DATA_BLOCK "EncoderET200S1COUNT_DB"   // DB87
// stored: AutoNumber true, InstanceOfName EncoderET200S1COUNT, OfSystemLibElement EncoderET200S1COUNT, OfSystemLibVersion 2.3
"EncoderET200S1COUNT"
   // VAR_INPUT
   //    EncErr : Bool;
   //    DOut_1 : Bool;
   //    DOut_2 : Bool;
   // END_VAR
   // VAR_OUTPUT
   //    DIn : Bool;
   // END_VAR
   // VAR_IN_OUT
   //    Axis : Struct
   //       Sample_T : Real;
   //       AxisType : Bool;
   //       EncoderType : Bool;
   //       Sim : Bool;
   //       AxisLimitMax : Real;
   //       AxisLimitMin : Real;
   //       MaxVelocity : Real;
   //       MaxAcceleration : Real;
   //       MaxDeceleration : Real;
   //       MonTimeTargetAppr : Real;
   //       TargetRange : Real;
   //       StandstillRange : Real;
   //       MaxFollowingDist : Real;
   //       MonitorTargetAppr : Bool;
   //       SWLimitEnable : Bool;
   //       FactorP : Real;
   //       ManVelocity : Real;
   //       ManEnable : Bool;
   //       EmergencyDec : Real;
   //       InputModuleInAddr : Int;
   //       InputModuleOutAddr : Int;
   //       InputChannelNo : Int;
   //       StepsPerRev : DInt;
   //       DisplacementPerRev : Real;
   //       NumberRevs : Int;
   //       PolarityEncoder : Int;
   //       PositionOffset : DInt;
   //       OutputModuleOutAddr : Int;
   //       OutputModuleInAddr : Int;
   //       OutputChannelNo : Int;
   //       PolarityDrive : Int;
   //       DriveInputAtMaxVel : Real;
   //       OffsetCompensation : Real;
   //       DriveInputAt100 : Real;
   //       Override : Real;
   //       ActPosition : Real;
   //       FollowingDistance : Real;
   //       RemainingDistance : Real;
   //       NomVelocity : Real;
   //       ActVelocity : Real;
   //       Sync : Bool;
   //       Error : Bool;
   //       ErrorAck : Bool;
   //       AxisState : Int;
   //       Err : Struct
   //          SWLimitMinExceeded : Bool;
   //          SWLimitMaxExceeded : Bool;
   //          TargetErr : Bool;
   //          NoSync : Bool;
   //          DirectionErr : Bool;
   //          DataErr : Bool;
   //          StartErr : Bool;
   //          DistanceErr : Bool;
   //          MasterErr : Bool;
   //          bit09 : Bool;
   //          bit10 : Bool;
   //          bit11 : Bool;
   //          bit12 : Bool;
   //          bit13 : Bool;
   //          bit14 : Bool;
   //          bit15 : Bool;
   //          StoppedMotion : Bool;
   //          EnableDriveErr : Bool;
   //          FollowingDistErr : Bool;
   //          StandstillErr : Bool;
   //          TargetApproachErr : Bool;
   //          EncoderErr : Bool;
   //          OutputErr : Bool;
   //          ConfigErr : Bool;
   //          DriveErr : Bool;
   //          bit25 : Bool;
   //          bit26 : Bool;
   //          bit27 : Bool;
   //          bit28 : Bool;
   //          bit29 : Bool;
   //          bit30 : Bool;
   //          bit31 : Bool;
   //       END_STRUCT;
   //       Config : Struct
   //          Err_AxisLimit : Bool;
   //          Err_MaxVelocity : Bool;
   //          Err_MaxAcceleration : Bool;
   //          Err_MaxDeceleration : Bool;
   //          Err_MonTimeTargetAppr : Bool;
   //          Err_TargetRange : Bool;
   //          Err_StandstillRange : Bool;
   //          Err_MaxFollowingDist : Bool;
   //          Err_EmergencyDec : Bool;
   //          Err_StepsPerRev : Bool;
   //          Err_DisplacementPerRev : Bool;
   //          Err_NumberRevs : Bool;
   //          Err_PolarityEncoder : Bool;
   //          Err_PolarityDrive : Bool;
   //          Err_DriveInputAtMaxVel : Bool;
   //          Err_AxisLength : Bool;
   //          Err_EncoderRange : Bool;
   //          Err_MaxVelRotaryAxis : Bool;
   //          Err_DriveInputAt100 : Bool;
   //       END_STRUCT;
   //       EncoderValue : DInt;
   //       RefPoint : Real;
   //       OutVelocity : Real;
   //       LastNomPosition : Real;
   //       LastNomVelocity : Real;
   //       LastNomDeceleration : Real;
   //       InternalNomPosition : Real;
   //       InternalActPos : Real;
   //       InternalPosOffset : Real;
   //       aufl : Real;
   //       AchsLaenge : Real;
   //       AchsLaenge_DI : DInt;
   //       AbsGeberLaenge_DI : DInt;
   //       LageIstwert_DI : DInt;
   //       Coord : DInt;
   //       DoneRef : Bool;
   //       EinInitLaeuft : Bool;
   //       AusInitLaeuft : Bool;
   //       EinQuittungLaeuft : Bool;
   //       AusQuittungLaeuft : Bool;
   //       EintreiberFahrbereit : Bool;
   //       ExecRef : Int;
   //       VLastNomPosition : Real;
   //       VLastNomVelocity : Real;
   //       LastInternalPosOffset : Real;
   //       RundKorrektur : Real;
   //       LastRundKorrektur : Real;
   //       LengthUnit : String[4];
   //       InputModuleType : String[24];
   //       OutputModuleType : String[24];
   //       Init : Struct
   //          I0 : Bool;
   //          I1 : Bool;
   //          I2 : Bool;
   //          I3 : Bool;
   //          I4 : Bool;
   //          I5 : Bool;
   //          I6 : Bool;
   //          I7 : Bool;
   //          I8 : Bool;
   //          I9 : Bool;
   //          I10 : Bool;
   //          I11 : Bool;
   //          I12 : Bool;
   //          I13 : Bool;
   //          I14 : Bool;
   //          I15 : Bool;
   //          I16 : Bool;
   //          I17 : Bool;
   //          I18 : Bool;
   //          I19 : Bool;
   //          I20 : Bool;
   //          I21 : Bool;
   //          I22 : Bool;
   //          I23 : Bool;
   //          I24 : Bool;
   //          I25 : Bool;
   //          I26 : Bool;
   //          I27 : Bool;
   //          I28 : Bool;
   //          I29 : Bool;
   //          I30 : Bool;
   //          I31 : Bool;
   //       END_STRUCT;
   //    END_STRUCT;
   //    Init : Bool;
   // END_VAR
   // VAR RETAIN
   //    Status : Struct
   //       STS_LOAD : Bool;
   //       ERR_LOAD : Bool;
   //       RES_STS_A : Bool;
   //       ERR_ENCODER : Bool;
   //       ERR_DO2 : Bool;
   //       ERR_PARA : Bool;
   //       ERR_DO1 : Bool;
   //       ERR_24V : Bool;
   //       STS_GATE : Bool;
   //       STS_DI : Bool;
   //       bit18 : Bool;
   //       STS_DO1 : Bool;
   //       STS_DO2 : Bool;
   //       bit21 : Bool;
   //       STS_C_UP : Bool;
   //       STS_C_DN : Bool;
   //       STS_SYN : Bool;
   //       bit09 : Bool;
   //       bit10 : Bool;
   //       STS_CMP1 : Bool;
   //       STS_CMP2 : Bool;
   //       STS_OFLW : Bool;
   //       STS_UFLW : Bool;
   //       STS_ND : Bool;
   //       byte3 : Byte;
   //    END_STRUCT;
   //    GeberAlt_DI : DInt;
   //    Addr_ActPos_DI : Int;
   //    Addr_Status : Int;
   //    Addr_LoadVal_DI : Int;
   //    Addr_Steuer : Int;
   //    Richtungsanpassung : Int;
   //    v_Faktor : Real;
   //    MaxZahl : DInt;
   //    MaxZahlHalb : DInt;
   //    PASteuer : Word;
   //    RefPointInt : Real;
   //    LoadVal_DW : DWord;
   //    EncoderZustand : Int;
   //    RefZustand : Int;
   //    aufl : Real;
   //    EncErr_alt : Bool;
   //    Taktsynchron : Bool;
   // END_VAR
BEGIN
END_DATA_BLOCK

DATA_BLOCK "IEC_Timer_0_DB"   // DB31
// stored: AutoNumber true, InstanceOfName TON_SFB, OfSystemLibElement TON, OfSystemLibVersion 1.0
"TON_SFB"
   // VAR_INPUT
   //    IN : Bool;
   //    PT : Time;
   // END_VAR
   // VAR_OUTPUT
   //    Q : Bool;
   //    ET : Time;
   // END_VAR
   // VAR RETAIN
   //    STATE : Byte;
   //    STIME : Time;
   //    ATIME : Time;
   // END_VAR
BEGIN
END_DATA_BLOCK

DATA_BLOCK "IEC_Timer_0_DB_1"   // DB60
// stored: AutoNumber true, InstanceOfName TOF_SFB, OfSystemLibElement TOF, OfSystemLibVersion 1.0
"TOF_SFB"
   // VAR_INPUT
   //    IN : Bool;
   //    PT : Time;
   // END_VAR
   // VAR_OUTPUT
   //    Q : Bool;
   //    ET : Time;
   // END_VAR
   // VAR RETAIN
   //    STATE : Byte;
   //    STIME : Time;
   //    ATIME : Time;
   // END_VAR
BEGIN
END_DATA_BLOCK

DATA_BLOCK "IEC_Timer_0_DB_3"   // DB91
// stored: AutoNumber true, InstanceOfName TON_SFB, OfSystemLibElement TON, OfSystemLibVersion 1.0
"TON_SFB"
   // VAR_INPUT
   //    IN : Bool;
   //    PT : Time;
   // END_VAR
   // VAR_OUTPUT
   //    Q : Bool;
   //    ET : Time;
   // END_VAR
   // VAR RETAIN
   //    STATE : Byte;
   //    STIME : Time;
   //    ATIME : Time;
   // END_VAR
BEGIN
END_DATA_BLOCK

DATA_BLOCK "MC_Simulation_DB"   // DB99
// stored: AutoNumber true, InstanceOfName MC_Simulation, OfSystemLibElement MC_Simulation, OfSystemLibVersion 2.1
"MC_Simulation"
   // VAR_IN_OUT
   //    Axis : Struct
   //       Sample_T : Real;
   //       AxisType : Bool;
   //       EncoderType : Bool;
   //       Sim : Bool;
   //       AxisLimitMax : Real;
   //       AxisLimitMin : Real;
   //       MaxVelocity : Real;
   //       MaxAcceleration : Real;
   //       MaxDeceleration : Real;
   //       MonTimeTargetAppr : Real;
   //       TargetRange : Real;
   //       StandstillRange : Real;
   //       MaxFollowingDist : Real;
   //       MonitorTargetAppr : Bool;
   //       SWLimitEnable : Bool;
   //       FactorP : Real;
   //       ManVelocity : Real;
   //       ManEnable : Bool;
   //       EmergencyDec : Real;
   //       InputModuleInAddr : Int;
   //       InputModuleOutAddr : Int;
   //       InputChannelNo : Int;
   //       StepsPerRev : DInt;
   //       DisplacementPerRev : Real;
   //       NumberRevs : Int;
   //       PolarityEncoder : Int;
   //       PositionOffset : DInt;
   //       OutputModuleOutAddr : Int;
   //       OutputModuleInAddr : Int;
   //       OutputChannelNo : Int;
   //       PolarityDrive : Int;
   //       DriveInputAtMaxVel : Real;
   //       OffsetCompensation : Real;
   //       DriveInputAt100 : Real;
   //       Override : Real;
   //       ActPosition : Real;
   //       FollowingDistance : Real;
   //       RemainingDistance : Real;
   //       NomVelocity : Real;
   //       ActVelocity : Real;
   //       Sync : Bool;
   //       Error : Bool;
   //       ErrorAck : Bool;
   //       AxisState : Int;
   //       Err : Struct
   //          SWLimitMinExceeded : Bool;
   //          SWLimitMaxExceeded : Bool;
   //          TargetErr : Bool;
   //          NoSync : Bool;
   //          DirectionErr : Bool;
   //          DataErr : Bool;
   //          StartErr : Bool;
   //          DistanceErr : Bool;
   //          MasterErr : Bool;
   //          bit09 : Bool;
   //          bit10 : Bool;
   //          bit11 : Bool;
   //          bit12 : Bool;
   //          bit13 : Bool;
   //          bit14 : Bool;
   //          bit15 : Bool;
   //          StoppedMotion : Bool;
   //          EnableDriveErr : Bool;
   //          FollowingDistErr : Bool;
   //          StandstillErr : Bool;
   //          TargetApproachErr : Bool;
   //          EncoderErr : Bool;
   //          OutputErr : Bool;
   //          ConfigErr : Bool;
   //          DriveErr : Bool;
   //          bit25 : Bool;
   //          bit26 : Bool;
   //          bit27 : Bool;
   //          bit28 : Bool;
   //          bit29 : Bool;
   //          bit30 : Bool;
   //          bit31 : Bool;
   //       END_STRUCT;
   //       Config : Struct
   //          Err_AxisLimit : Bool;
   //          Err_MaxVelocity : Bool;
   //          Err_MaxAcceleration : Bool;
   //          Err_MaxDeceleration : Bool;
   //          Err_MonTimeTargetAppr : Bool;
   //          Err_TargetRange : Bool;
   //          Err_StandstillRange : Bool;
   //          Err_MaxFollowingDist : Bool;
   //          Err_EmergencyDec : Bool;
   //          Err_StepsPerRev : Bool;
   //          Err_DisplacementPerRev : Bool;
   //          Err_NumberRevs : Bool;
   //          Err_PolarityEncoder : Bool;
   //          Err_PolarityDrive : Bool;
   //          Err_DriveInputAtMaxVel : Bool;
   //          Err_AxisLength : Bool;
   //          Err_EncoderRange : Bool;
   //          Err_MaxVelRotaryAxis : Bool;
   //          Err_DriveInputAt100 : Bool;
   //       END_STRUCT;
   //       EncoderValue : DInt;
   //       RefPoint : Real;
   //       OutVelocity : Real;
   //       LastNomPosition : Real;
   //       LastNomVelocity : Real;
   //       LastNomDeceleration : Real;
   //       InternalNomPosition : Real;
   //       InternalActPos : Real;
   //       InternalPosOffset : Real;
   //       aufl : Real;
   //       AchsLaenge : Real;
   //       AchsLaenge_DI : DInt;
   //       AbsGeberLaenge_DI : DInt;
   //       LageIstwert_DI : DInt;
   //       Coord : DInt;
   //       DoneRef : Bool;
   //       EinInitLaeuft : Bool;
   //       AusInitLaeuft : Bool;
   //       EinQuittungLaeuft : Bool;
   //       AusQuittungLaeuft : Bool;
   //       EintreiberFahrbereit : Bool;
   //       ExecRef : Int;
   //       VLastNomPosition : Real;
   //       VLastNomVelocity : Real;
   //       LastInternalPosOffset : Real;
   //       RundKorrektur : Real;
   //       LastRundKorrektur : Real;
   //       LengthUnit : String[4];
   //       InputModuleType : String[24];
   //       OutputModuleType : String[24];
   //       Init : Struct
   //          I0 : Bool;
   //          I1 : Bool;
   //          I2 : Bool;
   //          I3 : Bool;
   //          I4 : Bool;
   //          I5 : Bool;
   //          I6 : Bool;
   //          I7 : Bool;
   //          I8 : Bool;
   //          I9 : Bool;
   //          I10 : Bool;
   //          I11 : Bool;
   //          I12 : Bool;
   //          I13 : Bool;
   //          I14 : Bool;
   //          I15 : Bool;
   //          I16 : Bool;
   //          I17 : Bool;
   //          I18 : Bool;
   //          I19 : Bool;
   //          I20 : Bool;
   //          I21 : Bool;
   //          I22 : Bool;
   //          I23 : Bool;
   //          I24 : Bool;
   //          I25 : Bool;
   //          I26 : Bool;
   //          I27 : Bool;
   //          I28 : Bool;
   //          I29 : Bool;
   //          I30 : Bool;
   //          I31 : Bool;
   //       END_STRUCT;
   //    END_STRUCT;
   //    Init : Bool;
   // END_VAR
   // VAR RETAIN
   //    Raster : Bool;
   //    Bitanzahl : Int;
   //    LageDiff_R : Real;
   //    Faktor : Real;
   //    AusFaktor : Real;
   //    WertBei10V : Real;
   // END_VAR
BEGIN
END_DATA_BLOCK

DATA_BLOCK "Move2Done"   // DB88
// stored: AutoNumber true, InstanceOfName TON_SFB, OfSystemLibElement TON, OfSystemLibVersion 1.0
"TON_SFB"
   // VAR_INPUT
   //    IN : Bool;
   //    PT : Time;
   // END_VAR
   // VAR_OUTPUT
   //    Q : Bool;
   //    ET : Time;
   // END_VAR
   // VAR RETAIN
   //    STATE : Byte;
   //    STIME : Time;
   //    ATIME : Time;
   // END_VAR
BEGIN
END_DATA_BLOCK

DATA_BLOCK "NotEnoughProducts"   // DB84
// stored: AutoNumber true, InstanceOfName TON_SFB, OfSystemLibElement TON, OfSystemLibVersion 1.0
"TON_SFB"
   // VAR_INPUT
   //    IN : Bool;
   //    PT : Time;
   // END_VAR
   // VAR_OUTPUT
   //    Q : Bool;
   //    ET : Time;
   // END_VAR
   // VAR RETAIN
   //    STATE : Byte;
   //    STIME : Time;
   //    ATIME : Time;
   // END_VAR
BEGIN
END_DATA_BLOCK

DATA_BLOCK "OutputSinamics_DB"   // DB14
// stored: AutoNumber true, InstanceOfName OutputSinamics, OfSystemLibElement OutputSinamics, OfSystemLibVersion 2.3
"OutputSinamics"
   // VAR_INPUT
   //    TelNumber : Int;
   //    EnableDrive : Bool;
   //    StopMode : Int;
   //    OutErr : Bool;
   // END_VAR
   // VAR_OUTPUT
   //    OperationEnabled : Bool;
   //    Err_ID : Word;
   // END_VAR
   // VAR_IN_OUT
   //    Axis : Struct
   //       Sample_T : Real;
   //       AxisType : Bool;
   //       EncoderType : Bool;
   //       Sim : Bool;
   //       AxisLimitMax : Real;
   //       AxisLimitMin : Real;
   //       MaxVelocity : Real;
   //       MaxAcceleration : Real;
   //       MaxDeceleration : Real;
   //       MonTimeTargetAppr : Real;
   //       TargetRange : Real;
   //       StandstillRange : Real;
   //       MaxFollowingDist : Real;
   //       MonitorTargetAppr : Bool;
   //       SWLimitEnable : Bool;
   //       FactorP : Real;
   //       ManVelocity : Real;
   //       ManEnable : Bool;
   //       EmergencyDec : Real;
   //       InputModuleInAddr : Int;
   //       InputModuleOutAddr : Int;
   //       InputChannelNo : Int;
   //       StepsPerRev : DInt;
   //       DisplacementPerRev : Real;
   //       NumberRevs : Int;
   //       PolarityEncoder : Int;
   //       PositionOffset : DInt;
   //       OutputModuleOutAddr : Int;
   //       OutputModuleInAddr : Int;
   //       OutputChannelNo : Int;
   //       PolarityDrive : Int;
   //       DriveInputAtMaxVel : Real;
   //       OffsetCompensation : Real;
   //       DriveInputAt100 : Real;
   //       Override : Real;
   //       ActPosition : Real;
   //       FollowingDistance : Real;
   //       RemainingDistance : Real;
   //       NomVelocity : Real;
   //       ActVelocity : Real;
   //       Sync : Bool;
   //       Error : Bool;
   //       ErrorAck : Bool;
   //       AxisState : Int;
   //       Err : Struct
   //          SWLimitMinExceeded : Bool;
   //          SWLimitMaxExceeded : Bool;
   //          TargetErr : Bool;
   //          NoSync : Bool;
   //          DirectionErr : Bool;
   //          DataErr : Bool;
   //          StartErr : Bool;
   //          DistanceErr : Bool;
   //          MasterErr : Bool;
   //          bit09 : Bool;
   //          bit10 : Bool;
   //          bit11 : Bool;
   //          bit12 : Bool;
   //          bit13 : Bool;
   //          bit14 : Bool;
   //          bit15 : Bool;
   //          StoppedMotion : Bool;
   //          EnableDriveErr : Bool;
   //          FollowingDistErr : Bool;
   //          StandstillErr : Bool;
   //          TargetApproachErr : Bool;
   //          EncoderErr : Bool;
   //          OutputErr : Bool;
   //          ConfigErr : Bool;
   //          DriveErr : Bool;
   //          bit25 : Bool;
   //          bit26 : Bool;
   //          bit27 : Bool;
   //          bit28 : Bool;
   //          bit29 : Bool;
   //          bit30 : Bool;
   //          bit31 : Bool;
   //       END_STRUCT;
   //       Config : Struct
   //          Err_AxisLimit : Bool;
   //          Err_MaxVelocity : Bool;
   //          Err_MaxAcceleration : Bool;
   //          Err_MaxDeceleration : Bool;
   //          Err_MonTimeTargetAppr : Bool;
   //          Err_TargetRange : Bool;
   //          Err_StandstillRange : Bool;
   //          Err_MaxFollowingDist : Bool;
   //          Err_EmergencyDec : Bool;
   //          Err_StepsPerRev : Bool;
   //          Err_DisplacementPerRev : Bool;
   //          Err_NumberRevs : Bool;
   //          Err_PolarityEncoder : Bool;
   //          Err_PolarityDrive : Bool;
   //          Err_DriveInputAtMaxVel : Bool;
   //          Err_AxisLength : Bool;
   //          Err_EncoderRange : Bool;
   //          Err_MaxVelRotaryAxis : Bool;
   //          Err_DriveInputAt100 : Bool;
   //       END_STRUCT;
   //       EncoderValue : DInt;
   //       RefPoint : Real;
   //       OutVelocity : Real;
   //       LastNomPosition : Real;
   //       LastNomVelocity : Real;
   //       LastNomDeceleration : Real;
   //       InternalNomPosition : Real;
   //       InternalActPos : Real;
   //       InternalPosOffset : Real;
   //       aufl : Real;
   //       AchsLaenge : Real;
   //       AchsLaenge_DI : DInt;
   //       AbsGeberLaenge_DI : DInt;
   //       LageIstwert_DI : DInt;
   //       Coord : DInt;
   //       DoneRef : Bool;
   //       EinInitLaeuft : Bool;
   //       AusInitLaeuft : Bool;
   //       EinQuittungLaeuft : Bool;
   //       AusQuittungLaeuft : Bool;
   //       EintreiberFahrbereit : Bool;
   //       ExecRef : Int;
   //       VLastNomPosition : Real;
   //       VLastNomVelocity : Real;
   //       LastInternalPosOffset : Real;
   //       RundKorrektur : Real;
   //       LastRundKorrektur : Real;
   //       LengthUnit : String[4];
   //       InputModuleType : String[24];
   //       OutputModuleType : String[24];
   //       Init : Struct
   //          I0 : Bool;
   //          I1 : Bool;
   //          I2 : Bool;
   //          I3 : Bool;
   //          I4 : Bool;
   //          I5 : Bool;
   //          I6 : Bool;
   //          I7 : Bool;
   //          I8 : Bool;
   //          I9 : Bool;
   //          I10 : Bool;
   //          I11 : Bool;
   //          I12 : Bool;
   //          I13 : Bool;
   //          I14 : Bool;
   //          I15 : Bool;
   //          I16 : Bool;
   //          I17 : Bool;
   //          I18 : Bool;
   //          I19 : Bool;
   //          I20 : Bool;
   //          I21 : Bool;
   //          I22 : Bool;
   //          I23 : Bool;
   //          I24 : Bool;
   //          I25 : Bool;
   //          I26 : Bool;
   //          I27 : Bool;
   //          I28 : Bool;
   //          I29 : Bool;
   //          I30 : Bool;
   //          I31 : Bool;
   //       END_STRUCT;
   //    END_STRUCT;
   //    Init : Bool;
   // END_VAR
   // VAR RETAIN
   //    CONFIGURATION_DATA : Struct
   //       InputModuleInAddr : Int;
   //       OutputModuleOutAddr : Int;
   //       ProfiBus : Bool;
   //       ProfiNet : Bool;
   //       ID_Mastersystem : Int;
   //       Telegrammnumber : Int;
   //       TelegrFromInput : Int;
   //       InputFound : Bool;
   //       synchronous : Bool;
   //       invalid : Bool;
   //    END_STRUCT;
   //    Faktor : Real;
   //    OutputValue_R : Real;
   //    Lifecounter : Int;
   //    Addr_STW1 : Int;
   //    Addr_STW2 : Int;
   //    Addr_MRED : Int;
   //    Addr_ZSW1 : Int;
   //    Addr_ZSW2 : Int;
   //    Addr_MELDW : Int;
   //    Addr_NSOLL_B : Int;
   //    Addr_XERR : Int;
   //    Addr_KPC : Int;
   //    STW1_Offset : Int;
   //    STW2_Offset : Int;
   //    ZSW1_Offset : Int;
   //    ZSW2_Offset : Int;
   //    MRED_Offset : Int;
   //    MELDW_Offset : Int;
   //    NSOLL_B_Offset : Int;
   //    XERR_Offset : Int;
   //    KPC_Offset : Int;
   //    OutputValue : DInt;
   //    Quittungsautomat : Int;
   //    Einschaltautomat : Int;
   //    ZSW1 : Word;
   //    ZSW2 : Word;
   //    STW1 : Word;
   //    STW2 : Word;
   //    MELDW : Word;
   //    MRED : Word;
   //    wrong_OB : Bool;
   //    ERRORCODE : DWord;
   //    Virgin : Bool;
   //    FirstNormalRun : Bool;
   // END_VAR
BEGIN
END_DATA_BLOCK

DATA_BLOCK "OutputUniversal_DB"   // DB9
// stored: AutoNumber true, InstanceOfName OutputUniversal, OfSystemLibElement OutputUniversal, OfSystemLibVersion 2.1
"OutputUniversal"
   // VAR_INPUT
   //    EnableDrive : Bool;
   //    IntAtMaxVelocity : Int;
   //    OutErr : Bool;
   // END_VAR
   // VAR_OUTPUT
   //    OutputValue : Int;
   //    OutValAbs : Int;
   //    OutValSign : Bool;
   // END_VAR
   // VAR_IN_OUT
   //    Axis : Struct
   //       Sample_T : Real;
   //       AxisType : Bool;
   //       EncoderType : Bool;
   //       Sim : Bool;
   //       AxisLimitMax : Real;
   //       AxisLimitMin : Real;
   //       MaxVelocity : Real;
   //       MaxAcceleration : Real;
   //       MaxDeceleration : Real;
   //       MonTimeTargetAppr : Real;
   //       TargetRange : Real;
   //       StandstillRange : Real;
   //       MaxFollowingDist : Real;
   //       MonitorTargetAppr : Bool;
   //       SWLimitEnable : Bool;
   //       FactorP : Real;
   //       ManVelocity : Real;
   //       ManEnable : Bool;
   //       EmergencyDec : Real;
   //       InputModuleInAddr : Int;
   //       InputModuleOutAddr : Int;
   //       InputChannelNo : Int;
   //       StepsPerRev : DInt;
   //       DisplacementPerRev : Real;
   //       NumberRevs : Int;
   //       PolarityEncoder : Int;
   //       PositionOffset : DInt;
   //       OutputModuleOutAddr : Int;
   //       OutputModuleInAddr : Int;
   //       OutputChannelNo : Int;
   //       PolarityDrive : Int;
   //       DriveInputAtMaxVel : Real;
   //       OffsetCompensation : Real;
   //       DriveInputAt100 : Real;
   //       Override : Real;
   //       ActPosition : Real;
   //       FollowingDistance : Real;
   //       RemainingDistance : Real;
   //       NomVelocity : Real;
   //       ActVelocity : Real;
   //       Sync : Bool;
   //       Error : Bool;
   //       ErrorAck : Bool;
   //       AxisState : Int;
   //       Err : Struct
   //          SWLimitMinExceeded : Bool;
   //          SWLimitMaxExceeded : Bool;
   //          TargetErr : Bool;
   //          NoSync : Bool;
   //          DirectionErr : Bool;
   //          DataErr : Bool;
   //          StartErr : Bool;
   //          DistanceErr : Bool;
   //          MasterErr : Bool;
   //          bit09 : Bool;
   //          bit10 : Bool;
   //          bit11 : Bool;
   //          bit12 : Bool;
   //          bit13 : Bool;
   //          bit14 : Bool;
   //          bit15 : Bool;
   //          StoppedMotion : Bool;
   //          EnableDriveErr : Bool;
   //          FollowingDistErr : Bool;
   //          StandstillErr : Bool;
   //          TargetApproachErr : Bool;
   //          EncoderErr : Bool;
   //          OutputErr : Bool;
   //          ConfigErr : Bool;
   //          DriveErr : Bool;
   //          bit25 : Bool;
   //          bit26 : Bool;
   //          bit27 : Bool;
   //          bit28 : Bool;
   //          bit29 : Bool;
   //          bit30 : Bool;
   //          bit31 : Bool;
   //       END_STRUCT;
   //       Config : Struct
   //          Err_AxisLimit : Bool;
   //          Err_MaxVelocity : Bool;
   //          Err_MaxAcceleration : Bool;
   //          Err_MaxDeceleration : Bool;
   //          Err_MonTimeTargetAppr : Bool;
   //          Err_TargetRange : Bool;
   //          Err_StandstillRange : Bool;
   //          Err_MaxFollowingDist : Bool;
   //          Err_EmergencyDec : Bool;
   //          Err_StepsPerRev : Bool;
   //          Err_DisplacementPerRev : Bool;
   //          Err_NumberRevs : Bool;
   //          Err_PolarityEncoder : Bool;
   //          Err_PolarityDrive : Bool;
   //          Err_DriveInputAtMaxVel : Bool;
   //          Err_AxisLength : Bool;
   //          Err_EncoderRange : Bool;
   //          Err_MaxVelRotaryAxis : Bool;
   //          Err_DriveInputAt100 : Bool;
   //       END_STRUCT;
   //       EncoderValue : DInt;
   //       RefPoint : Real;
   //       OutVelocity : Real;
   //       LastNomPosition : Real;
   //       LastNomVelocity : Real;
   //       LastNomDeceleration : Real;
   //       InternalNomPosition : Real;
   //       InternalActPos : Real;
   //       InternalPosOffset : Real;
   //       aufl : Real;
   //       AchsLaenge : Real;
   //       AchsLaenge_DI : DInt;
   //       AbsGeberLaenge_DI : DInt;
   //       LageIstwert_DI : DInt;
   //       Coord : DInt;
   //       DoneRef : Bool;
   //       EinInitLaeuft : Bool;
   //       AusInitLaeuft : Bool;
   //       EinQuittungLaeuft : Bool;
   //       AusQuittungLaeuft : Bool;
   //       EintreiberFahrbereit : Bool;
   //       ExecRef : Int;
   //       VLastNomPosition : Real;
   //       VLastNomVelocity : Real;
   //       LastInternalPosOffset : Real;
   //       RundKorrektur : Real;
   //       LastRundKorrektur : Real;
   //       LengthUnit : String[4];
   //       InputModuleType : String[24];
   //       OutputModuleType : String[24];
   //       Init : Struct
   //          I0 : Bool;
   //          I1 : Bool;
   //          I2 : Bool;
   //          I3 : Bool;
   //          I4 : Bool;
   //          I5 : Bool;
   //          I6 : Bool;
   //          I7 : Bool;
   //          I8 : Bool;
   //          I9 : Bool;
   //          I10 : Bool;
   //          I11 : Bool;
   //          I12 : Bool;
   //          I13 : Bool;
   //          I14 : Bool;
   //          I15 : Bool;
   //          I16 : Bool;
   //          I17 : Bool;
   //          I18 : Bool;
   //          I19 : Bool;
   //          I20 : Bool;
   //          I21 : Bool;
   //          I22 : Bool;
   //          I23 : Bool;
   //          I24 : Bool;
   //          I25 : Bool;
   //          I26 : Bool;
   //          I27 : Bool;
   //          I28 : Bool;
   //          I29 : Bool;
   //          I30 : Bool;
   //          I31 : Bool;
   //       END_STRUCT;
   //    END_STRUCT;
   //    Init : Bool;
   // END_VAR
   // VAR RETAIN
   //    Velo2Volt : Real;
   //    Volt2Int : Real;
   // END_VAR
BEGIN
END_DATA_BLOCK

DATA_BLOCK "ProductBufferTimer"   // DB80
// stored: AutoNumber true, InstanceOfName TON_SFB, OfSystemLibElement TON, OfSystemLibVersion 1.0
"TON_SFB"
   // VAR_INPUT
   //    IN : Bool;
   //    PT : Time;
   // END_VAR
   // VAR_OUTPUT
   //    Q : Bool;
   //    ET : Time;
   // END_VAR
   // VAR RETAIN
   //    STATE : Byte;
   //    STIME : Time;
   //    ATIME : Time;
   // END_VAR
BEGIN
END_DATA_BLOCK

DATA_BLOCK "ProductCounter"   // DB21
// stored: AutoNumber true, InstanceOfName CTU_SFB, OfSystemLibElement CTU, OfSystemLibVersion 1.0
"CTU_SFB"
   // VAR_INPUT
   //    CU : Bool;
   //    R : Bool;
   //    PV : Int;
   // END_VAR
   // VAR_OUTPUT
   //    Q : Bool;
   //    CV : Int;
   // END_VAR
   // VAR RETAIN
   //    CUO : Bool;
   // END_VAR
BEGIN
END_DATA_BLOCK

DATA_BLOCK "RestAferReferenceRun"   // DB52
// stored: AutoNumber true, InstanceOfName TON_SFB, OfSystemLibElement TON, OfSystemLibVersion 1.0
"TON_SFB"
   // VAR_INPUT
   //    IN : Bool;
   //    PT : Time;
   // END_VAR
   // VAR_OUTPUT
   //    Q : Bool;
   //    ET : Time;
   // END_VAR
   // VAR RETAIN
   //    STATE : Byte;
   //    STIME : Time;
   //    ATIME : Time;
   // END_VAR
BEGIN
END_DATA_BLOCK

DATA_BLOCK "SafetyTimer"   // DB16
// stored: AutoNumber true, InstanceOfName TON_SFB, OfSystemLibElement TON, OfSystemLibVersion 1.0
"TON_SFB"
   // VAR_INPUT
   //    IN : Bool;
   //    PT : Time;
   // END_VAR
   // VAR_OUTPUT
   //    Q : Bool;
   //    ET : Time;
   // END_VAR
   // VAR RETAIN
   //    STATE : Byte;
   //    STIME : Time;
   //    ATIME : Time;
   // END_VAR
BEGIN
END_DATA_BLOCK

DATA_BLOCK "StartDelayTimer"   // DB57
// stored: AutoNumber true, InstanceOfName TON_SFB, OfSystemLibElement TON, OfSystemLibVersion 1.0
"TON_SFB"
   // VAR_INPUT
   //    IN : Bool;
   //    PT : Time;
   // END_VAR
   // VAR_OUTPUT
   //    Q : Bool;
   //    ET : Time;
   // END_VAR
   // VAR RETAIN
   //    STATE : Byte;
   //    STIME : Time;
   //    ATIME : Time;
   // END_VAR
BEGIN
END_DATA_BLOCK

DATA_BLOCK "TimerOffDelayMove2"   // DB97
// stored: AutoNumber true, InstanceOfName TOF_SFB, OfSystemLibElement TOF, OfSystemLibVersion 1.0
"TOF_SFB"
   // VAR_INPUT
   //    IN : Bool;
   //    PT : Time;
   // END_VAR
   // VAR_OUTPUT
   //    Q : Bool;
   //    ET : Time;
   // END_VAR
   // VAR RETAIN
   //    STATE : Byte;
   //    STIME : Time;
   //    ATIME : Time;
   // END_VAR
BEGIN
END_DATA_BLOCK

DATA_BLOCK "Timer_0_5s"   // DB30
// stored: AutoNumber true, InstanceOfName TON_SFB, OfSystemLibElement TON, OfSystemLibVersion 1.0
"TON_SFB"
   // VAR_INPUT
   //    IN : Bool;
   //    PT : Time;
   // END_VAR
   // VAR_OUTPUT
   //    Q : Bool;
   //    ET : Time;
   // END_VAR
   // VAR RETAIN
   //    STATE : Byte;
   //    STIME : Time;
   //    ATIME : Time;
   // END_VAR
BEGIN
END_DATA_BLOCK

DATA_BLOCK "Timer_Aanvoerband"   // DB7
// stored: AutoNumber true, InstanceOfName TON_SFB, OfSystemLibElement TON, OfSystemLibVersion 1.0
"TON_SFB"
   // VAR_INPUT
   //    IN : Bool;
   //    PT : Time;
   // END_VAR
   // VAR_OUTPUT
   //    Q : Bool;
   //    ET : Time;
   // END_VAR
   // VAR RETAIN
   //    STATE : Byte;
   //    STIME : Time;
   //    ATIME : Time;
   // END_VAR
BEGIN
END_DATA_BLOCK

DATA_BLOCK "Timer_AxisCheck"   // DB40
// stored: AutoNumber true, InstanceOfName TON_SFB, OfSystemLibElement TON, OfSystemLibVersion 1.0
"TON_SFB"
   // VAR_INPUT
   //    IN : Bool;
   //    PT : Time;
   // END_VAR
   // VAR_OUTPUT
   //    Q : Bool;
   //    ET : Time;
   // END_VAR
   // VAR RETAIN
   //    STATE : Byte;
   //    STIME : Time;
   //    ATIME : Time;
   // END_VAR
BEGIN
END_DATA_BLOCK

DATA_BLOCK "Timer_ProductInterval"   // DB20
// stored: AutoNumber true, InstanceOfName TON_SFB, OfSystemLibElement TON, OfSystemLibVersion 1.0
"TON_SFB"
   // VAR_INPUT
   //    IN : Bool;
   //    PT : Time;
   // END_VAR
   // VAR_OUTPUT
   //    Q : Bool;
   //    ET : Time;
   // END_VAR
   // VAR RETAIN
   //    STATE : Byte;
   //    STIME : Time;
   //    ATIME : Time;
   // END_VAR
BEGIN
END_DATA_BLOCK

DATA_BLOCK "Timer_Retourband"   // DB70
// stored: AutoNumber true, InstanceOfName TON_SFB, OfSystemLibElement TON, OfSystemLibVersion 1.0
"TON_SFB"
   // VAR_INPUT
   //    IN : Bool;
   //    PT : Time;
   // END_VAR
   // VAR_OUTPUT
   //    Q : Bool;
   //    ET : Time;
   // END_VAR
   // VAR RETAIN
   //    STATE : Byte;
   //    STIME : Time;
   //    ATIME : Time;
   // END_VAR
BEGIN
END_DATA_BLOCK

DATA_BLOCK "Timer_Retourband_Off"   // DB72
// stored: AutoNumber true, InstanceOfName TOF_SFB, OfSystemLibElement TOF, OfSystemLibVersion 1.0
"TOF_SFB"
   // VAR_INPUT
   //    IN : Bool;
   //    PT : Time;
   // END_VAR
   // VAR_OUTPUT
   //    Q : Bool;
   //    ET : Time;
   // END_VAR
   // VAR RETAIN
   //    STATE : Byte;
   //    STIME : Time;
   //    ATIME : Time;
   // END_VAR
BEGIN
END_DATA_BLOCK

DATA_BLOCK "Timer_Signal_1"   // DB36
// stored: AutoNumber true, InstanceOfName TP_SFB, OfSystemLibElement TP, OfSystemLibVersion 1.0
"TP_SFB"
   // VAR_INPUT
   //    IN : Bool;
   //    PT : Time;
   // END_VAR
   // VAR_OUTPUT
   //    Q : Bool;
   //    ET : Time;
   // END_VAR
   // VAR RETAIN
   //    STATE : Byte;
   //    STIME : Time;
   //    ATIME : Time;
   // END_VAR
BEGIN
END_DATA_BLOCK

DATA_BLOCK "Timer_Signal_2"   // DB37
// stored: AutoNumber true, InstanceOfName TON_SFB, OfSystemLibElement TON, OfSystemLibVersion 1.0
"TON_SFB"
   // VAR_INPUT
   //    IN : Bool;
   //    PT : Time;
   // END_VAR
   // VAR_OUTPUT
   //    Q : Bool;
   //    ET : Time;
   // END_VAR
   // VAR RETAIN
   //    STATE : Byte;
   //    STIME : Time;
   //    ATIME : Time;
   // END_VAR
BEGIN
END_DATA_BLOCK

DATA_BLOCK "Timer_Trilgoten"   // DB5
// stored: AutoNumber true, InstanceOfName TON_SFB, OfSystemLibElement TON, OfSystemLibVersion 1.0
"TON_SFB"
   // VAR_INPUT
   //    IN : Bool;
   //    PT : Time;
   // END_VAR
   // VAR_OUTPUT
   //    Q : Bool;
   //    ET : Time;
   // END_VAR
   // VAR RETAIN
   //    STATE : Byte;
   //    STIME : Time;
   //    ATIME : Time;
   // END_VAR
BEGIN
END_DATA_BLOCK

DATA_BLOCK "TotalProductsCounter"   // DB22
// stored: AutoNumber true, InstanceOfName CTU_SFB, OfSystemLibElement CTU, OfSystemLibVersion 1.0
"CTU_SFB"
   // VAR_INPUT
   //    CU : Bool;
   //    R : Bool;
   //    PV : Int;
   // END_VAR
   // VAR_OUTPUT
   //    Q : Bool;
   //    CV : Int;
   // END_VAR
   // VAR RETAIN
   //    CUO : Bool;
   // END_VAR
BEGIN
END_DATA_BLOCK

DATA_BLOCK "Uitlooptimer_Aanvoerband"   // DB10
// stored: AutoNumber true, InstanceOfName TON_SFB, OfSystemLibElement TON, OfSystemLibVersion 1.0
"TON_SFB"
   // VAR_INPUT
   //    IN : Bool;
   //    PT : Time;
   // END_VAR
   // VAR_OUTPUT
   //    Q : Bool;
   //    ET : Time;
   // END_VAR
   // VAR RETAIN
   //    STATE : Byte;
   //    STIME : Time;
   //    ATIME : Time;
   // END_VAR
BEGIN
END_DATA_BLOCK

DATA_BLOCK "Uitlooptimer_Trilgoten"   // DB11
// stored: AutoNumber true, InstanceOfName TON_SFB, OfSystemLibElement TON, OfSystemLibVersion 1.0
"TON_SFB"
   // VAR_INPUT
   //    IN : Bool;
   //    PT : Time;
   // END_VAR
   // VAR_OUTPUT
   //    Q : Bool;
   //    ET : Time;
   // END_VAR
   // VAR RETAIN
   //    STATE : Byte;
   //    STIME : Time;
   //    ATIME : Time;
   // END_VAR
BEGIN
END_DATA_BLOCK

DATA_BLOCK "WarningTimer2"   // DB32
// stored: AutoNumber true, InstanceOfName TON_SFB, OfSystemLibElement TON, OfSystemLibVersion 1.0
"TON_SFB"
   // VAR_INPUT
   //    IN : Bool;
   //    PT : Time;
   // END_VAR
   // VAR_OUTPUT
   //    Q : Bool;
   //    ET : Time;
   // END_VAR
   // VAR RETAIN
   //    STATE : Byte;
   //    STIME : Time;
   //    ATIME : Time;
   // END_VAR
BEGIN
END_DATA_BLOCK

DATA_BLOCK "WarningTimer3"   // DB61
// stored: AutoNumber true, InstanceOfName TON_SFB, OfSystemLibElement TON, OfSystemLibVersion 1.0
"TON_SFB"
   // VAR_INPUT
   //    IN : Bool;
   //    PT : Time;
   // END_VAR
   // VAR_OUTPUT
   //    Q : Bool;
   //    ET : Time;
   // END_VAR
   // VAR RETAIN
   //    STATE : Byte;
   //    STIME : Time;
   //    ATIME : Time;
   // END_VAR
BEGIN
END_DATA_BLOCK

DATA_BLOCK "Blinker_SimulateSensor_DB"   // DB100
VERSION : 0.1
// stored: AutoNumber true, InstanceOfName Blinker, InstanceOfType FB
"Blinker"
BEGIN
END_DATA_BLOCK

DATA_BLOCK "Blinker_Yellow"   // DB102
VERSION : 0.1
// stored: AutoNumber true, InstanceOfName Blinker, InstanceOfType FB
"Blinker"
BEGIN
END_DATA_BLOCK

DATA_BLOCK "ConfirimationDrive1Timer"   // DB101
// stored: AutoNumber true, InstanceOfName TON_SFB, OfSystemLibElement TON, OfSystemLibVersion 1.0
"TON_SFB"
   // VAR_INPUT
   //    IN : Bool;
   //    PT : Time;
   // END_VAR
   // VAR_OUTPUT
   //    Q : Bool;
   //    ET : Time;
   // END_VAR
   // VAR RETAIN
   //    STATE : Byte;
   //    STIME : Time;
   //    ATIME : Time;
   // END_VAR
BEGIN
END_DATA_BLOCK
